(* IEC 61131-3 sources: AXOpen/src/components.cognex.vision/ctrl/src/AxoInsight/v_6_0_0/TypeStructuresAndEnums, 19 files *)

(* ---- AxoInsight_AcquisitionControl.st ---- *)
NAMESPACE AXOpen.Components.Cognex.Vision.v_6_0_0_0
    TYPE
        {#ix-attr:[Container(Layout.Wrap)]}
        AxoInsight_AcquisitionControl :
        STRUCT
            {#ix-set:AttributeName = "<#Trigger enable#>"}
            TriggerEnable 			:	BOOL;
            {#ix-set:AttributeName = "<#Trigger#>"}
            Trigger					:	BOOL;
            {#ix-set:AttributeName = "<#Clear exposure complete#>"}
            ClearExposureComplete :  BOOL;
            {#ix-set:AttributeName = "<#Set offline#>"}
            SetOffline :  BOOL;
        END_STRUCT;
    END_TYPE
END_NAMESPACE

(* ---- AxoInsight_AcquisitionStatus.st ---- *)
NAMESPACE AXOpen.Components.Cognex.Vision.v_6_0_0_0
    TYPE
        {#ix-attr:[Container(Layout.Wrap)]}
        AxoInsight_AcquisitionStatus :
        STRUCT
            {#ix-set:AttributeName = "<#Trigger ready#>"}
            TriggerReady 		:	BOOL;
            {#ix-set:AttributeName = "<#Trigger acknowledge#>"}
            TriggerAcknowledge 	:	BOOL;
            {#ix-set:AttributeName = "<#Exposure complete#>"}
            ExposureComplete	:	BOOL;
            {#ix-set:AttributeName = "<#Missed acquisition#>"}
            MissedAcquisition 	:	BOOL;
            {#ix-set:AttributeName = "<#Offline reason 0#>"}
            OfflineReason0      :   BOOL;
            {#ix-set:AttributeName = "<#Offline reason 1#>"}
            OfflineReason1      :   BOOL;
            {#ix-set:AttributeName = "<#Offline reason 2#>"}
            OfflineReason2      :   BOOL;
            {#ix-set:AttributeName = "<#Online#>"}
            Online              :   BOOL;
            {#ix-set:AttributeName = "<#Acquisition ID#>"}
            AcquisitionID       :   UINT;
        END_STRUCT;
    END_TYPE
END_NAMESPACE

(* ---- AxoInsight_CommandControl.st ---- *)
NAMESPACE AXOpen.Components.Cognex.Vision.v_6_0_0_0
    TYPE
        {#ix-attr:[Container(Layout.Wrap)]}
        {S7.extern=ReadWrite}
        AxoInsight_CommandControl :
        STRUCT
            {#ix-set:AttributeName = "<#Command#>"}
            Command        : UINT;
        END_STRUCT;
    END_TYPE
END_NAMESPACE

(* ---- AxoInsight_CommandStatus.st ---- *)
NAMESPACE AXOpen.Cognex.Vision.v_6_0_0_0
    TYPE
        {#ix-attr:[Container(Layout.Wrap)]}
        AxoInsight_CommandStatus :
        STRUCT
            {#ix-set:AttributeName = "<#Current job ID#>"}
            CurrentJobID  : UINT;
        END_STRUCT;
    END_TYPE
END_NAMESPACE

(* ---- AxoInsight_Config.st ---- *)
NAMESPACE AXOpen.Components.Cognex.Vision.v_6_0_0_0
    TYPE
        {#ix-attr:[Container(Layout.Wrap)]}
        {S7.extern=ReadWrite}
        AxoInsight_Config :
        STRUCT
            {#ix-set:AttributeName = "<#Info time#>"}
            InfoTime : LTIME := LT#10S;
            {#ix-set:AttributeName = "<#Error time#>"}
            ErrorTime : LTIME := LT#50S;
            {#ix-set:AttributeName = "<#Task timeout#>"}
            TaskTimeout : LTIME := LT#50S;
            {#ix-set:AttributeName = "<#Max job number#>"}
            MaxJobNumber : UINT := UINT#999;
            {#ix-set:AttributeName = "<#Result data size#>"}
            ResultDataSize : UINT;
            {#ix-set:AttributeName = "<#User data size#>"}
            UserDataSize : UINT;
        END_STRUCT;
    END_TYPE
END_NAMESPACE

(* ---- AxoInsight_InspectionControl.st ---- *)
NAMESPACE AXOpen.Components.Cognex.Vision.v_6_0_0_0
    TYPE
        {#ix-attr:[Container(Layout.Wrap)]}
        AxoInsight_InspectionControl :
        STRUCT
            {#ix-set:AttributeName = "<#Enable results buffering#>"}
            EnableResultsBuffering          :   BOOL;
            {#ix-set:AttributeName = "<#Acknowledge inspection results#>"}
            AcknowledgeInspectionResults    :   BOOL;
            {#ix-set:AttributeName = "<#Extended user data set#>"}
            ExtendedUserDataSet             :   BOOL;
            {#ix-set:AttributeName = "<#Execute command#>"}
            ExecuteCommand                  :   BOOL;
            {#ix-set:AttributeName = "<#Clear error#>"}
            ClearError                      :   BOOL;
        END_STRUCT;
    END_TYPE
END_NAMESPACE

(* ---- AxoInsight_InspectionStatus.st ---- *)
NAMESPACE AXOpen.Components.Cognex.Vision.v_6_0_0_0
    TYPE
        {#ix-attr:[Container(Layout.Wrap)]}
        AxoInsight_InspectionStatus :
        STRUCT
            {#ix-set:AttributeName = "<#System busy#>"}
            SystemBusy                      :   BOOL;
            {#ix-set:AttributeName = "<#Inspection completed#>"}
            InspectionCompleted             :   BOOL;
            {#ix-set:AttributeName = "<#Results buffer overrun#>"}
            ResultsBufferOverrun            :   BOOL;
            {#ix-set:AttributeName = "<#Results valid#>"}
            ResultsValid                    :   BOOL;
            {#ix-set:AttributeName = "<#Command executing#>"}
            CommandExecuting                :   BOOL;
            {#ix-set:AttributeName = "<#Command complete#>"}
            CommandComplete                 :   BOOL;
            {#ix-set:AttributeName = "<#Command failed#>"}
            CommandFailed                   :   BOOL;
            {#ix-set:AttributeName = "<#Extended user data set acknowledge#>"}
            ExtendedUserDataSetAcknowledge  :   BOOL;
            {#ix-set:AttributeName = "<#Overall job pass fail#>"}
            OverallJobPassFail              :   BOOL;
            {#ix-set:AttributeName = "<#Test run ready#>"}
            TestRunReady                    :   BOOL;
            {#ix-set:AttributeName = "<#Error#>"}
            Error                           :   BOOL;
            {#ix-set:AttributeName = "<#Error code#>"}
            ErrorCode                       :   UINT;
        END_STRUCT;
    END_TYPE
END_NAMESPACE

(* ---- AxoInsight_Results.st ---- *)
NAMESPACE AXOpen.Cognex.Vision.v_6_0_0_0
    TYPE
        {#ix-attr:[Container(Layout.Wrap)]}
        AxoInsight_Results :
        STRUCT
            {#ix-set:AttributeName = "<#Inspection ID#>"}
            InspectionID : UINT;
            {#ix-set:AttributeName = "<#Result code#>"}
            ResultCode : UINT;
            // {#ix-set:AttributeName = "<#Inspection results#>"}
            // InspectionResults : AxoByteArray255;
        END_STRUCT;
    END_TYPE
END_NAMESPACE

(* ---- AxoInsight_SoftEventControl.st ---- *)
NAMESPACE AXOpen.Components.Cognex.Vision.v_6_0_0_0
    TYPE
        {#ix-attr:[Container(Layout.Wrap)]}
        {S7.extern=ReadWrite}
        AxoInsight_SoftEventControl :
        STRUCT
            {#ix-set:AttributeName = "<#Trigger soft-event#>"}
            TriggerSoftEvent : AxoBoolArray8;
        END_STRUCT;
    END_TYPE
END_NAMESPACE

(* ---- AxoInsight_SoftEventStatus.st ---- *)
NAMESPACE AXOpen.Components.Cognex.Vision.v_6_0_0_0
    TYPE
        {#ix-attr:[Container(Layout.Wrap)]}
        AxoInsight_SoftEventStatus :
        STRUCT
            {#ix-set:AttributeName = "<#Trigger soft-event acknowledge#>"}
            TriggerSoftEventAcknowledge : AxoBoolArray8;
        END_STRUCT;
    END_TYPE
END_NAMESPACE

(* ---- AxoInsight_User.st ---- *)
NAMESPACE AXOpen.Cognex.Vision.v_6_0_0_0
    TYPE
        {#ix-attr:[Container(Layout.Wrap)]}
        AxoInsight_User :
        STRUCT
            {#ix-set:AttributeName = "<#User data#>"}
            UserData : AxoByteArray255;
        END_STRUCT;
    END_TYPE
END_NAMESPACE

(* ---- eAxoInsight_ResultDataSize.st ---- *)
NAMESPACE AXOpen.Components.Cognex.Vision.v_6_0_0_0
    TYPE PUBLIC
        eAxoInsight_ResultDataSize : INT
        (
            RESULT_DATA_SIZE_INVALID := 0,
            RESULT_DATA_16B := 16,
            RESULT_DATA_32B := 32,
            RESULT_DATA_64B := 64,
            RESULT_DATA_128B := 128,
            RESULT_DATA_250B := 250
         ) := RESULT_DATA_64B;
    END_TYPE
END_NAMESPACE

(* ---- eAxoInsight_UserDataSize.st ---- *)
NAMESPACE AXOpen.Components.Cognex.Vision.v_6_0_0_0
    TYPE PUBLIC
        eAxoInsight_UserDataSize : INT
        (
            USER_DATA_SIZE_INVALID := 0,
            USER_DATA_16B := 16,
            USER_DATA_32B := 32,
            USER_DATA_64B := 64,
            USER_DATA_128B := 128,
            USER_DATA_254B := 254
         ) := USER_DATA_64B;
    END_TYPE
END_NAMESPACE

(* ---- AxoBoolArray8.st ---- *)
NAMESPACE AXOpen.Components.Cognex.Vision.v_6_0_0_0
    {S7.extern=ReadWrite}
    CLASS PUBLIC AxoBoolArray8 EXTENDS AXOpen.Core.AxoBoolArray
        VAR PUBLIC
            Data : ARRAY [0..7] OF BOOL;
        END_VAR
    END_CLASS
END_NAMESPACE

(* ---- AxoByteArray255.st ---- *)
NAMESPACE AXOpen.Cognex.Vision.v_6_0_0_0
    // TYPE
    //     AxoByteArray255 :
    //     STRUCT
    //         DataChanged : BOOL;
    //         Data : ARRAY [0..254] OF BYTE;
    //     END_STRUCT;
    // END_TYPE
    CLASS PUBLIC AxoByteArray255
        VAR PUBLIC
            DataChanged : BOOL;
            Data : ARRAY [0..254] OF BYTE;
        END_VAR
    END_CLASS
END_NAMESPACE

(* ---- AxoInsight_HWIDs.st ---- *)
NAMESPACE AXOpen.Components.Cognex.Vision.v_6_0_0_0
    {#ix-attr:[Container(Layout.Stack)]}
    {S7.extern=ReadWrite}
    CLASS PUBLIC AxoInsight_HWIDs
        VAR PUBLIC
            {#ix-set:AttributeName = "<#Hardware ID of the device#>"}
            HW_Device               :  UINT;
            {#ix-set:AttributeName = "<#Hardware ID of the 'AcquisitionControl' submodule#>"}
            HwIdAcquisitionControl  :   UINT;
            {#ix-set:AttributeName = "<#Hardware ID of the 'AcquisitionStatus' submodule#>"}
            HwIdAcquisitionStatus   :   UINT;
            {#ix-set:AttributeName = "<#Hardware ID of the 'InspectionControl' submodule#>"}
            HwIdInspectionControl      :   UINT;
            {#ix-set:AttributeName = "<#Hardware ID of the 'InspectionStatus' submodule#>"}
            HwIdInspectionStatus       :   UINT;
            {#ix-set:AttributeName = "<#Hardware ID of the 'CommandControl' submodule#>"}
            HwIdCommandControl    :   UINT;
            {#ix-set:AttributeName = "<#Hardware ID of the 'SoftEventControl' submodule#>"}
            HwIdSoftEventControl    :   UINT;
            {#ix-set:AttributeName = "<#Hardware ID of the 'UserData' submodule#>"}
            HwIdUserData            :   UINT;
            {#ix-set:AttributeName = "<#Hardware ID of the 'ResultData' submodule#>"}
            HwIdResultData          :   UINT;
        END_VAR
    END_CLASS
END_NAMESPACE

(* ---- AxoInsight_ResultData.st ---- *)
NAMESPACE AXOpen.Components.Cognex.Vision.v_6_0_0_0
    {S7.extern=ReadWrite}
    CLASS PUBLIC AxoInsight_ResultData EXTENDS AXOpen.Core.AxoByteArray
        VAR PUBLIC
            Data : ARRAY [0..249] OF BYTE;
        END_VAR
    END_CLASS
END_NAMESPACE

(* ---- AxoInsight_Status.st ---- *)
USING AXOpen.Core;
NAMESPACE AXOpen.Components.Cognex.Vision.v_6_0_0_0
    {#ix-attr:[Container(Layout.Stack)]}
    {S7.extern=ReadWrite}
    CLASS AxoInsight_Status EXTENDS AXOpen.Components.Abstractions.AxoComponent_Status
        VAR PUBLIC
            {#ix-attr:[Container(Layout.Wrap)]}
            {#ix-set:AttributeName = "<#Current job name#>"}
            CurrentJobName : STRING;
            {#ix-set:AttributeName = "<#Current job number#>"}
            CurrentJobNumber : UINT;
        END_VAR
    END_CLASS
END_NAMESPACE

(* ---- AxoInsight_UserData.st ---- *)
NAMESPACE AXOpen.Components.Cognex.Vision.v_6_0_0_0
    CLASS PUBLIC AxoInsight_UserData EXTENDS AXOpen.Core.AxoByteArray
        VAR PUBLIC
            Data : ARRAY [0..253] OF BYTE;
        END_VAR
    END_CLASS
END_NAMESPACE
